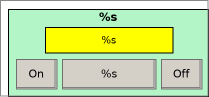
VISUALIZATION VISU_ECOMODE  // 209x97
    RoundedRectangle (8,9 201x88), "%s", text list: 'TextList_EcoMode', text index: 8
    RoundedRectangle (45,27 128x26), "%s", invisible if: NOT MACHINE.STATE_Standby, text list: 'TextList_EcoMode', text index: 10
    Button (62,59 94x30), "%s", text list: 'TextList_EcoMode', text index: 9
        OnMouseClick: change screen: VISU_CONFIG_ECOMODE
    Button (16,59 41x30), "On", invisible if: MACHINE.STATE_Standby, input disabled if: MACHINE.STATE_Prod
        toggle MACHINE.M_Standby
    Button (161,59 41x30), "Off", invisible if: NOT MACHINE.STATE_Standby, input disabled if: MACHINE.STATE_Prod
        toggle MACHINE.M_End_Standby
END_VISUALIZATION

(* stored: Version 1.1.0.1, ProductVersion 3.1.4024.11
   Visu VISU_ECOMODE: Id {ac6126f4-e219-43f5-875e-62a830a65432} *)
